(* CODESYS project Untitled1.project

Project tree, tasks and I/O mapping:
  Device : CODESYS Control Win V3, 3S - Smart Software Solutions GmbH, order no. 305021, version 3.5.11.30
    application Application
      libraries: Standard, * (System)
      task MainTask (cyclic, interval t#20ms, priority 1) calls PLC_PRG
      program PLC_PRG [SFC]: p1_active, P0_active, p2_active, p3_active
      program PRGM_LD [LD]
*)

// Device/Application/PLC_PRG
PROGRAM PLC_PRG
VAR
	b0: BOOL;
	b1: BOOL;
	b2: BOOL;
	pe: BOOL;
	pf: BOOL;
	
	fc0: BOOL := TRUE ;
	fc1: BOOL;
	fc2: BOOL;
	
	i1: BOOL;
	km1: BOOL;
	km2: BOOL;
	
	trig0: R_trig;
	T0: TOF;
	time0: TIME;
	
	T1: TOF;
	trig1: R_TRIG;
	time1: TIME;
	
	T2: TOF;
	trig2: R_TRIG;
	time2: TIME;
END_VAR

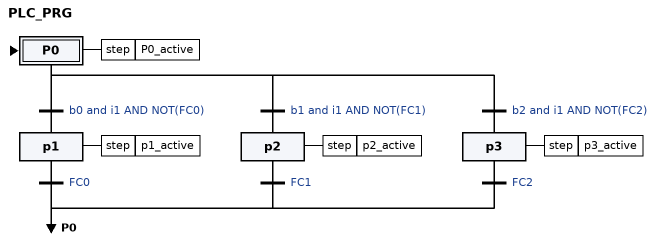
INITIAL_STEP P0:
    P0_active(N);  // step action
END_STEP
TRANSITION FROM P0 TO p1
    := b0 and i1 AND NOT(FC0);
END_TRANSITION
STEP p1:
    p1_active(N);  // step action
END_STEP
TRANSITION FROM p1 TO P0
    := FC0;
END_TRANSITION
TRANSITION FROM P0 TO p2
    := b1 and i1 AND NOT(FC1);
END_TRANSITION
STEP p2:
    p2_active(N);  // step action
END_STEP
TRANSITION FROM p2 TO P0
    := FC1;
END_TRANSITION
TRANSITION FROM P0 TO p3
    := b2 and i1 AND NOT(FC2);
END_TRANSITION
STEP p3:
    p3_active(N);  // step action
END_STEP
TRANSITION FROM p3 TO P0
    := FC2;
END_TRANSITION

ACTION p1_active:
trig0(clk:= b0);
T0(IN := trig0.Q, pt:= T#3S,ET=> TIME0);
IF NOT(T0.Q) THEN 
	km2 := TRUE;
END_IF

IF PE THEN 
	km2 := FALSE;
	km1 := FALSE;
END_IF
END_ACTION

ACTION P0_active:
KM1:= FALSE;
KM2:=FALSE;
END_ACTION

ACTION p2_active:
trig1(clk:= b1);
T1(IN := trig1.Q, pt:= T#3S,ET=> TIME1);
IF NOT(T1.Q) THEN 
	IF FC0 THEN 
		KM1:=TRUE;
	END_IF
	
	IF FC2 THEN 
		KM2:=TRUE;
	END_IF
END_IF

IF PE THEN 
	km2 := FALSE;
	km1 := FALSE;
END_IF
END_ACTION

ACTION p3_active:
trig2(clk:= b2);
T2(IN := trig2.Q, pt:= T#3S,ET=> TIME2);
IF NOT(T2.Q) THEN 
	KM1:=TRUE;
END_IF

IF PE THEN 
	km2 := FALSE;
	km1 := FALSE;
END_IF
END_ACTION

END_PROGRAM

// Device/Application/PRGM_LD
PROGRAM PRGM_LD
VAR
	b0: BOOL;
	b1: BOOL;
	b2: BOOL;
	pe: BOOL;
	pf: BOOL;
	
	fc0: BOOL := TRUE ;
	fc1: BOOL;
	fc2: BOOL;
	
	i1: BOOL;
	km1: BOOL;
	km2: BOOL;
	
	trig0: R_trig;
	T0: TOF;
	time0: TIME;
	
	T1: TOF;
	trig1: R_TRIG;
	time1: TIME;
	
	T2: TOF;
	trig2: R_TRIG;
	time2: TIME;
	
	P0: BOOL;
	P1: BOOL;
	P2: BOOL;
	P3: BOOL;
	
	TR1: BOOL;
	TR2: BOOL;
	TR3: BOOL;
	TR4: BOOL;
	TR5: BOOL;
	TR6: BOOL;
	
	CYCLE: BOOL;
	QTRIG0: BOOL;
	QTRIG1: BOOL;
	QTRIG2: BOOL;
	T0Q: BOOL;
	T1Q: BOOL;
	T2Q: BOOL;
END_VAR
VAR // added by the converter: edge detectors and wires of the graphical bodies
    _w1, _w2, _w3, _w4, _w5, _w6, _w7, _w8 : BOOL;
END_VAR

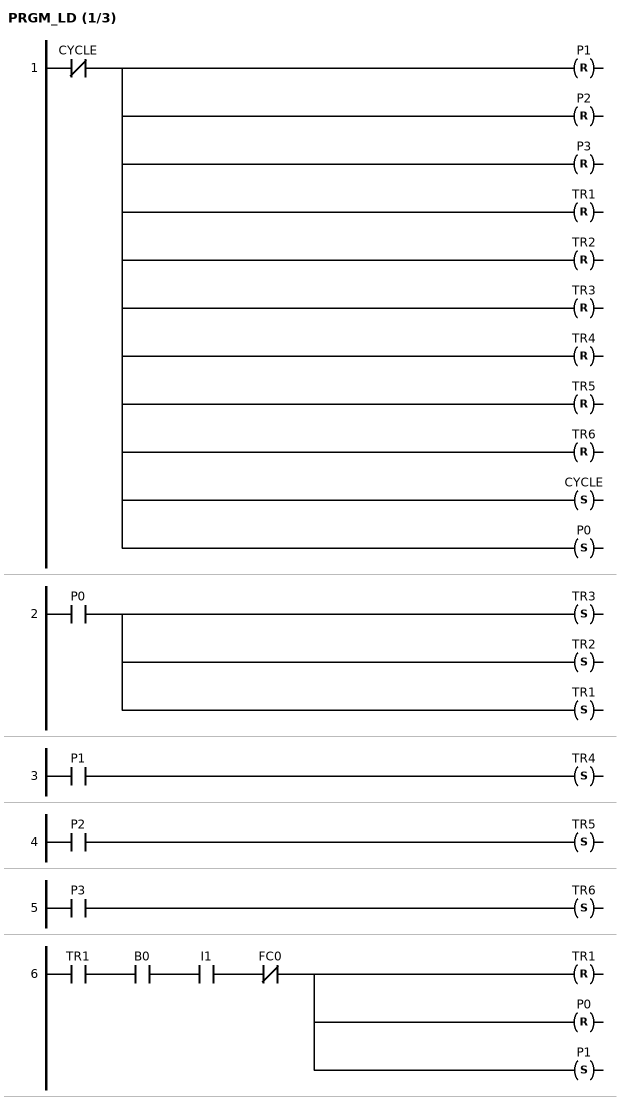
// NETWORK 1
_w1 := NOT CYCLE;
P1 R= _w1;
P2 R= _w1;
P3 R= _w1;
TR1 R= _w1;
TR2 R= _w1;
TR3 R= _w1;
TR4 R= _w1;
TR5 R= _w1;
TR6 R= _w1;
CYCLE S= _w1;
P0 S= _w1;

// NETWORK 2
TR3 S= P0;
TR2 S= P0;
TR1 S= P0;

// NETWORK 3
TR4 S= P1;

// NETWORK 4
TR5 S= P2;

// NETWORK 5
TR6 S= P3;

// NETWORK 6
_w2 := TR1 AND B0 AND I1 AND NOT FC0;
TR1 R= _w2;
P0 R= _w2;
P1 S= _w2;

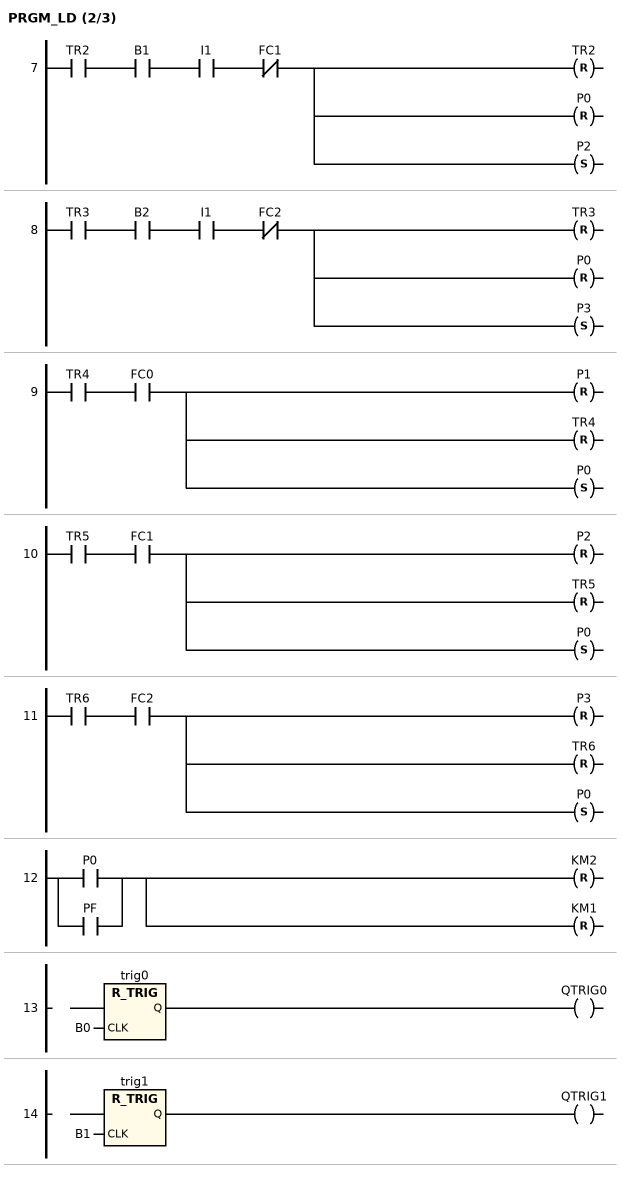
// NETWORK 7
_w3 := TR2 AND B1 AND I1 AND NOT FC1;
TR2 R= _w3;
P0 R= _w3;
P2 S= _w3;

// NETWORK 8
_w4 := TR3 AND B2 AND I1 AND NOT FC2;
TR3 R= _w4;
P0 R= _w4;
P3 S= _w4;

// NETWORK 9
_w5 := TR4 AND FC0;
P1 R= _w5;
TR4 R= _w5;
P0 S= _w5;

// NETWORK 10
_w6 := TR5 AND FC1;
P2 R= _w6;
TR5 R= _w6;
P0 S= _w6;

// NETWORK 11
_w7 := TR6 AND FC2;
P3 R= _w7;
TR6 R= _w7;
P0 S= _w7;

// NETWORK 12
_w8 := P0 OR PF;
KM2 R= _w8;
KM1 R= _w8;

// NETWORK 13
trig0(CLK := B0); // R_TRIG
QTRIG0 := trig0.Q;

// NETWORK 14
trig1(CLK := B1); // R_TRIG
QTRIG1 := trig1.Q;

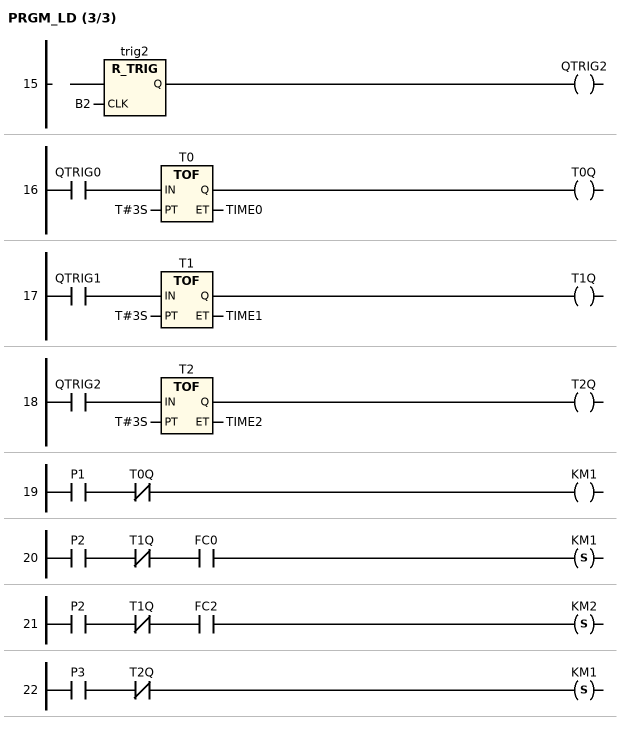
// NETWORK 15
trig2(CLK := B2); // R_TRIG
QTRIG2 := trig2.Q;

// NETWORK 16
T0(IN := QTRIG0, PT := T#3S, ET => TIME0); // TOF
T0Q := T0.Q;

// NETWORK 17
T1(IN := QTRIG1, PT := T#3S, ET => TIME1); // TOF
T1Q := T1.Q;

// NETWORK 18
T2(IN := QTRIG2, PT := T#3S, ET => TIME2); // TOF
T2Q := T2.Q;

// NETWORK 19
KM1 := P1 AND NOT T0Q;

// NETWORK 20
KM1 S= P2 AND NOT T1Q AND FC0;

// NETWORK 21
KM2 S= P2 AND NOT T1Q AND FC2;

// NETWORK 22
KM1 S= P3 AND NOT T2Q;

END_PROGRAM
